// TIA Portal V15.1 export
// export: Created 2020-06-12T07:35:45.2255859Z, ExportSetting None, DisplayName Totally Integrated Automation Portal, DisplayVersion V15.1, DisplayName TIA Portal Openness, DisplayVersion V15.1, DisplayName STEP 7 Professional, DisplayVersion V15.1, DisplayName STEP 7 Safety, DisplayVersion V15.1, DisplayName WinCC Advanced, DisplayVersion V15.1
FUNCTION "O2_meas" : Void   // FC128, FBD
{ S7_Optimized_Access := 'TRUE' }
// stored: SetENOAutomatically False
   VAR_TEMP
      tOxMeasOn : Bool;
      tOxMeasOff : Bool;
      tCleanOn : Bool;
      tCleanOff : Bool;
      tCheckAirOn : Bool;
      tCheckAirOff : Bool;
      tCheckNOn : Bool;
      tCheckNOff : Bool;
   END_VAR
   VAR_TEMP   // added for the SCL form of the ladder/FBD networks
      _w1 : Bool;
   END_VAR
BEGIN

REGION Network 1: HMI request treat
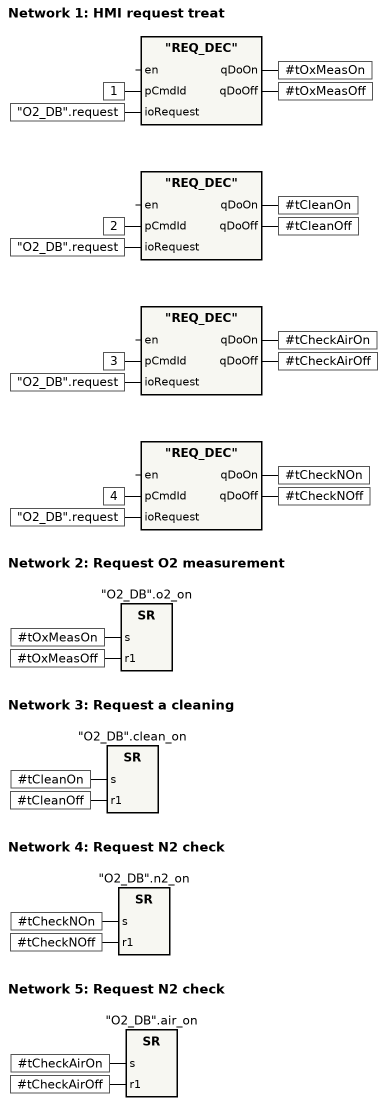
   "REQ_DEC"(pCmdId := 1, ioRequest := "O2_DB".request, qDoOn => #tOxMeasOn, qDoOff => #tOxMeasOff);
   "REQ_DEC"(pCmdId := 2, ioRequest := "O2_DB".request, qDoOn => #tCleanOn, qDoOff => #tCleanOff);
   "REQ_DEC"(pCmdId := 3, ioRequest := "O2_DB".request, qDoOn => #tCheckAirOn, qDoOff => #tCheckAirOff);
   "REQ_DEC"(pCmdId := 4, ioRequest := "O2_DB".request, qDoOn => #tCheckNOn, qDoOff => #tCheckNOff);
END_REGION

REGION Network 2: Request O2 measurement
   IF #tOxMeasOn THEN
       "O2_DB".o2_on := TRUE;   // SR flip-flop
   END_IF;
   IF #tOxMeasOff THEN "O2_DB".o2_on := FALSE; END_IF;
END_REGION

REGION Network 3: Request a cleaning
   IF #tCleanOn THEN
       "O2_DB".clean_on := TRUE;   // SR flip-flop
   END_IF;
   IF #tCleanOff THEN "O2_DB".clean_on := FALSE; END_IF;
END_REGION

REGION Network 4: Request N2 check
   IF #tCheckNOn THEN
       "O2_DB".n2_on := TRUE;   // SR flip-flop
   END_IF;
   IF #tCheckNOff THEN "O2_DB".n2_on := FALSE; END_IF;
END_REGION

REGION Network 5: Request N2 check
   IF #tCheckAirOn THEN
       "O2_DB".air_on := TRUE;   // SR flip-flop
   END_IF;
   IF #tCheckAirOff THEN "O2_DB".air_on := FALSE; END_IF;
END_REGION

REGION Network 6: Deactivate other requests
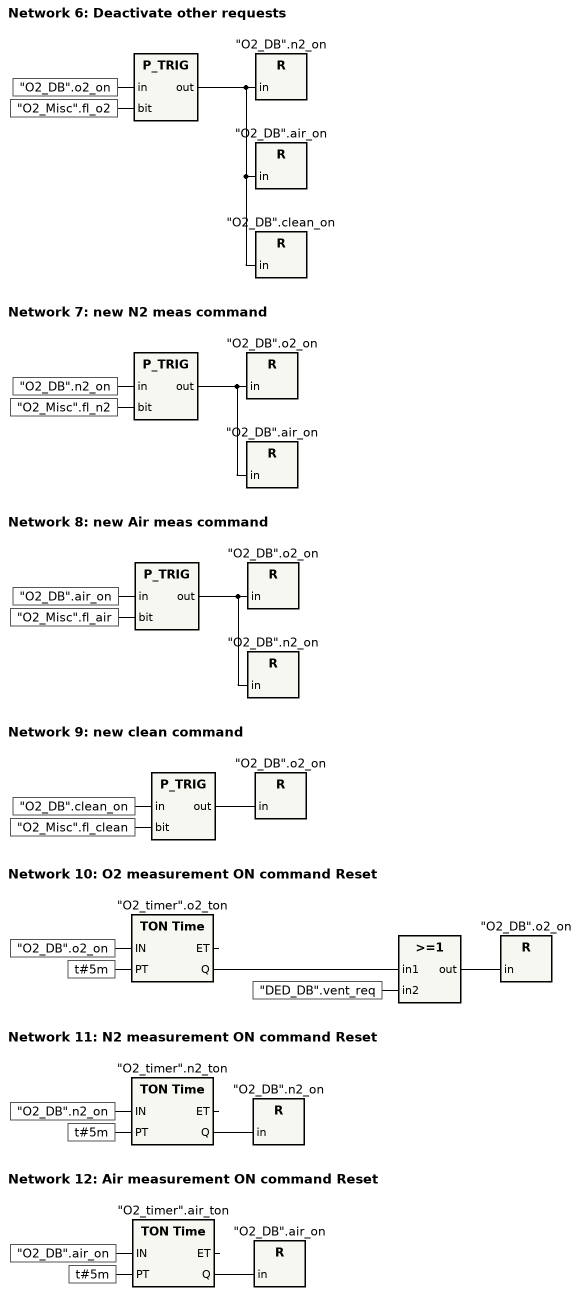
   #_w1 := "O2_DB".o2_on AND NOT "O2_Misc".fl_o2;   // rising edge
   "O2_Misc".fl_o2 := "O2_DB".o2_on;
   IF #_w1 THEN
       "O2_DB".n2_on := FALSE;
       "O2_DB".air_on := FALSE;
       "O2_DB".clean_on := FALSE;
   END_IF;
END_REGION

REGION Network 7: new N2 meas command
   #_w1 := "O2_DB".n2_on AND NOT "O2_Misc".fl_n2;   // rising edge
   "O2_Misc".fl_n2 := "O2_DB".n2_on;
   IF #_w1 THEN
       "O2_DB".o2_on := FALSE;
       "O2_DB".air_on := FALSE;
   END_IF;
END_REGION

REGION Network 8: new Air meas command
   #_w1 := "O2_DB".air_on AND NOT "O2_Misc".fl_air;   // rising edge
   "O2_Misc".fl_air := "O2_DB".air_on;
   IF #_w1 THEN
       "O2_DB".o2_on := FALSE;
       "O2_DB".n2_on := FALSE;
   END_IF;
END_REGION

REGION Network 9: new clean command
   #_w1 := "O2_DB".clean_on AND NOT "O2_Misc".fl_clean;   // rising edge
   "O2_Misc".fl_clean := "O2_DB".clean_on;
   IF #_w1 THEN "O2_DB".o2_on := FALSE; END_IF;
END_REGION

REGION Network 10: O2 measurement ON command Reset
   "O2_timer".o2_ton.TON(IN := "O2_DB".o2_on, PT := t#5m);
   IF "O2_timer".o2_ton.Q OR "DED_DB".vent_req THEN "O2_DB".o2_on := FALSE; END_IF;
END_REGION

REGION Network 11: N2 measurement ON command Reset
   "O2_timer".n2_ton.TON(IN := "O2_DB".n2_on, PT := t#5m);
   IF "O2_timer".n2_ton.Q THEN "O2_DB".n2_on := FALSE; END_IF;
END_REGION

REGION Network 12: Air measurement ON command Reset
   "O2_timer".air_ton.TON(IN := "O2_DB".air_on, PT := t#5m);
   IF "O2_timer".air_ton.Q THEN "O2_DB".air_on := FALSE; END_IF;
END_REGION

REGION Network 13: Clean ON command Reset
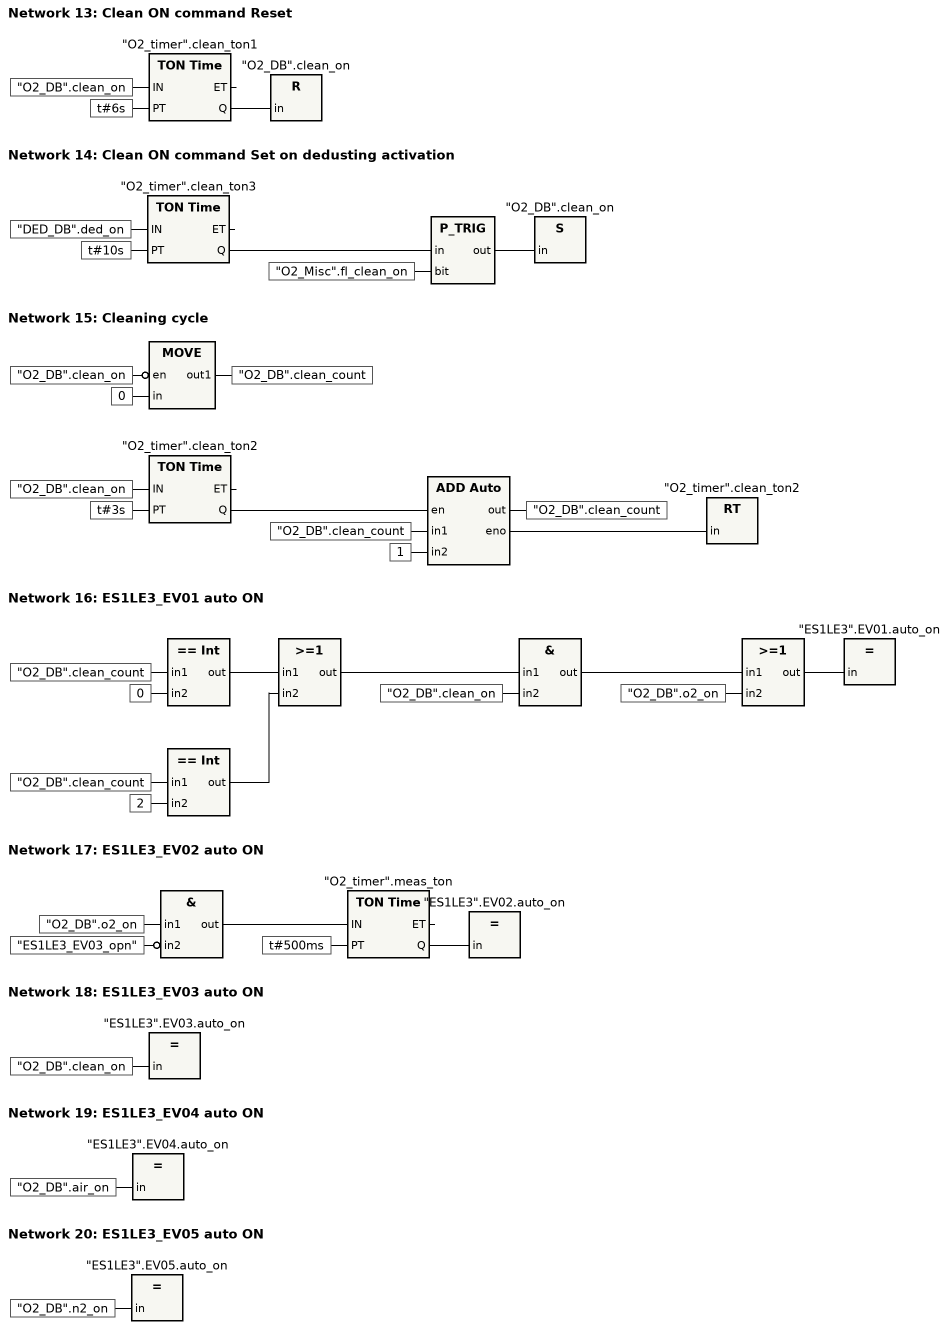
   "O2_timer".clean_ton1.TON(IN := "O2_DB".clean_on, PT := t#6s);
   IF "O2_timer".clean_ton1.Q THEN "O2_DB".clean_on := FALSE; END_IF;
END_REGION

REGION Network 14: Clean ON command Set on dedusting activation
   "O2_timer".clean_ton3.TON(IN := "DED_DB".ded_on, PT := t#10s);
   #_w1 := "O2_timer".clean_ton3.Q AND NOT "O2_Misc".fl_clean_on;   // rising edge
   "O2_Misc".fl_clean_on := "O2_timer".clean_ton3.Q;
   IF #_w1 THEN "O2_DB".clean_on := TRUE; END_IF;
END_REGION

REGION Network 15: Cleaning cycle
   IF NOT "O2_DB".clean_on THEN "O2_DB".clean_count := 0; END_IF;
   "O2_timer".clean_ton2.TON(IN := "O2_DB".clean_on, PT := t#3s);
   IF "O2_timer".clean_ton2.Q THEN
       "O2_DB".clean_count := "O2_DB".clean_count + 1;
       RESET_TIMER("O2_timer".clean_ton2);
   END_IF;
END_REGION

REGION Network 16: ES1LE3_EV01 auto ON
   "ES1LE3".EV01.auto_on := ((("O2_DB".clean_count = 0) OR ("O2_DB".clean_count = 2)) AND "O2_DB".clean_on) OR "O2_DB".o2_on;
END_REGION

REGION Network 17: ES1LE3_EV02 auto ON
   "O2_timer".meas_ton.TON(IN := "O2_DB".o2_on AND NOT "ES1LE3_EV03_opn", PT := t#500ms);
   "ES1LE3".EV02.auto_on := "O2_timer".meas_ton.Q;
END_REGION

REGION Network 18: ES1LE3_EV03 auto ON
   "ES1LE3".EV03.auto_on := "O2_DB".clean_on;
END_REGION

REGION Network 19: ES1LE3_EV04 auto ON
   "ES1LE3".EV04.auto_on := "O2_DB".air_on;
END_REGION

REGION Network 20: ES1LE3_EV05 auto ON
   "ES1LE3".EV05.auto_on := "O2_DB".n2_on;
END_REGION

REGION Network 21: ES1LE3_M02 auto ON
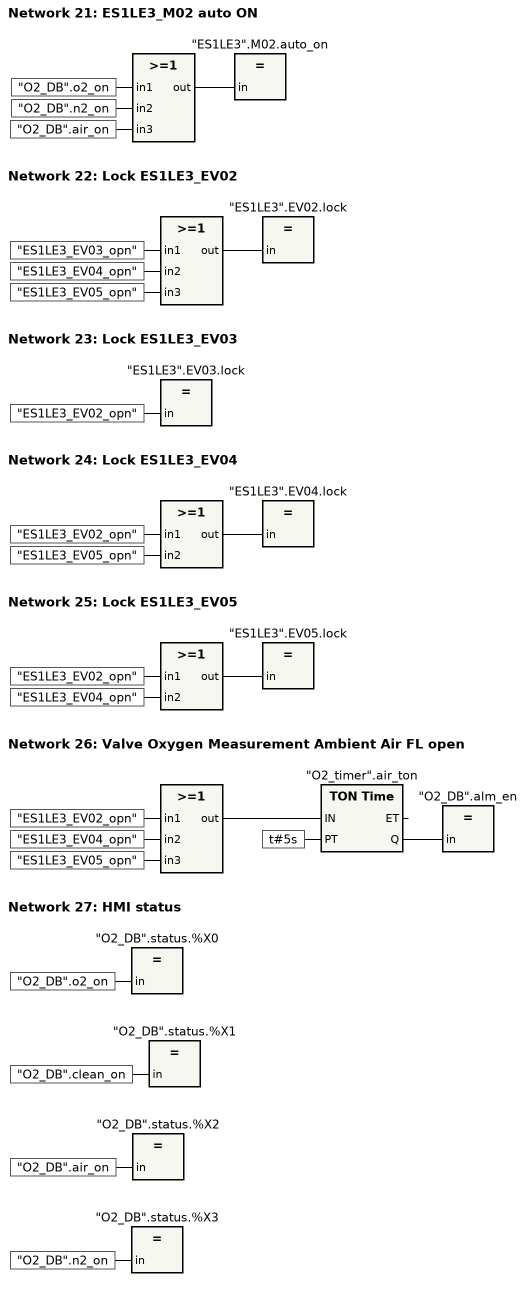
   "ES1LE3".M02.auto_on := "O2_DB".o2_on OR "O2_DB".n2_on OR "O2_DB".air_on;
END_REGION

REGION Network 22: Lock ES1LE3_EV02
   "ES1LE3".EV02.lock := "ES1LE3_EV03_opn" OR "ES1LE3_EV04_opn" OR "ES1LE3_EV05_opn";
END_REGION

REGION Network 23: Lock ES1LE3_EV03
   "ES1LE3".EV03.lock := "ES1LE3_EV02_opn";
END_REGION

REGION Network 24: Lock ES1LE3_EV04
   "ES1LE3".EV04.lock := "ES1LE3_EV02_opn" OR "ES1LE3_EV05_opn";
END_REGION

REGION Network 25: Lock ES1LE3_EV05
   "ES1LE3".EV05.lock := "ES1LE3_EV02_opn" OR "ES1LE3_EV04_opn";
END_REGION

REGION Network 26: Valve Oxygen Measurement Ambient Air FL open
   "O2_timer".air_ton.TON(IN := "ES1LE3_EV02_opn" OR "ES1LE3_EV04_opn" OR "ES1LE3_EV05_opn", PT := t#5s);
   "O2_DB".alm_en := "O2_timer".air_ton.Q;
END_REGION

REGION Network 27: HMI status
   "O2_DB".status.%X0 := "O2_DB".o2_on;
   "O2_DB".status.%X1 := "O2_DB".clean_on;
   "O2_DB".status.%X2 := "O2_DB".air_on;
   "O2_DB".status.%X3 := "O2_DB".n2_on;
END_REGION
END_FUNCTION
